FUNCTION_BLOCK Test_TStreamAdd_Read_INT EXTENDS TUnitTestBase
VAR
    Stream : TStream(StreamLength := 2);
END_VAR



Stream.Init(2);

Stream.Add_INT(1234);
    
Assertion.AssertEquals_UDINT(
    Expected := 2,
    Actual := Stream.Position,
    VariableName := 'Stream.Position');
    
Stream.Seek(0);

Assertion.AssertEquals_INT(
    Expected := 1234,
    Actual := Stream.Read_INT(),
    VariableName := 'Stream.Read_INT()');
    
Assertion.AssertEquals_UDINT(
    Expected := 2,
    Actual := Stream.Position,
    VariableName := 'Stream.Position');
    
    
TestFinished();

END_FUNCTION_BLOCK

(* stored: Version 1.1.0.1, ProductVersion 3.1.4024.4
   POU Test_TStreamAdd_Read_INT: Id {0a9e8abd-ccb7-4985-a0ed-3a7360014937}, SpecialFunc None *)
